// Mitsubishi GX Works2 project: bmov01   PLC: Q02/Q02H

PROGRAM MAIN
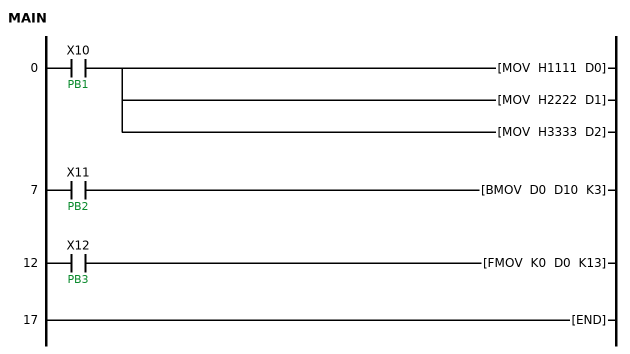
0     LD      X10  ; PB1
      MOV     H1111 D0
      MOV     H2222 D1
      MOV     H3333 D2
7     LD      X11  ; PB2
      BMOV    D0 D10 K3
12    LD      X12  ; PB3
      FMOV    K0 D0 K13
17    END
END_PROGRAM

// device comments not shown above
X0  ; 공급_후
X1  ; 공급_전
X2  ; 드릴_상
X3  ; 드릴_하
X4  ; 송출_후
X5  ; 송출_전
X6  ; 배출_후
X7  ; 배출_전
X8  ; 매거진
X9  ; 비금속
X0A  ; 금속
Y20  ; 공급_전
Y21  ; 공급_후
Y22  ; 드릴_하강
Y23  ; 송출_전
Y24  ; 송출_후
Y25  ; 배출_전
Y26  ; 배출_후
Y27  ; 컨베어
Y28  ; 가공드
Y29  ; 적색
Y2A  ; 황색
Y2B  ; 녹색
